(* CoDeSys 2.3 export: EXPORTEDPROJECT.EXP *)
(* Libraries: STANDARD.LIB 5.6.98 13:03:02 *)

(* Task configuration *)
TASK Standard (PRIORITY := 0, INTERVAL := T#10ms);
MAIN
END_TASK

(* POU MAIN, SFC *)
PROGRAM MAIN
VAR
	SRullo_presenza AT%IX0.0:BOOL;
	SRullo_Finecorsa AT%IX0.1:BOOL;
	SAsc_Altezza AT%IX0.2:BOOL;
	SRullo_Pistoneavanti AT%IX0.3:BOOL;
	SAsc_Capacitivo AT%IX0.4:BOOL;
	SAsc_Soglia AT%IX0.5:BOOL;
	SAsc_Pistonedietro AT%IX0.6:BOOL;
	SAsc_Basso AT%IX0.7:BOOL;
	SAsc_Alto AT%IX0.8:BOOL;
         SGiostra_Colore AT %IX0.9:BOOL;
	SGiostra_Altezza AT%IX1.0:BOOL;
	SGiostra_PresenzaPinza AT%IX1.1:BOOL;
	SDremel_alto AT%IX1.2:BOOL;
	SDremel_Basso AT %IX1.3:BOOL;
	SGiostra_Presenza AT %IX1.4:BOOL;
	SGiostra_AltezzaAlto AT %IX1.5:BOOL;
	SGiostra_AltezzaBasso AT %IX1.6:BOOL;
	SGiostra_MarkerAlto AT%IX1.7: BOOL;
	SGiostra_MarkerBasso AT%IX1.8: BOOL;



	AAsc_salita AT%QX0.0:BOOL;
	AAsc_discesa AT%QX0.1:BOOL;
	AAsc_aria AT%QX0.2:BOOL;
	AAsc_pistone AT %QX0.3:BOOL;
	ARullo_pistone AT %QX0.4:BOOL;
	ARullo_avanti AT %QX0.5:BOOL;
	AGiostra_Pistone AT %QX0.6:BOOL;
	AGiostra_Marker AT%QX4.0:BOOL;
	AGiostra_Gira AT %QX0.8:BOOL;
	AGiostra_Scarta AT%QX2.9:BOOL;
         AGiostra_Dremel AT%QX1.3:BOOL;
	AGiostra_AbbassaDremel AT%QX1.1:BOOL;
	AGiostra_Altezza AT%QX1.2:BOOL;

	S_RC_FineCorsaBasso AT %IX8.0:BOOL;
	S_RC_FineCorsaAlto AT %IX8.1:BOOL;
	S_RC_FineCorsaDestra AT %IX8.2:BOOL;
	S_RC_FineCorsaSinistra AT %IX8.3:BOOL;
	S_RC_PresenzaPinza AT %IX8.4:BOOL;
	S_RC_PinzaSensore AT %IX8.5:BOOL;
	S_RC_ScivoloPieno AT %IX8.7:BOOL;

	S_RC_Encoder AT %IX8.6:BOOL;
	S_RC_Estensimetro AT %IW2:WORD;

	A_RC_MovBasso AT %QX8.0:BOOL;
	A_RC_MovAlto AT %QX8.1:BOOL;
	A_RC_MovDestra AT %QX8.2:BOOL;
	A_RC_MovSinistra AT %QX8.3:BOOL;
	A_RC_Pinza AT %QX8.4:BOOL;

	T1: TON;
	T2: TON;
	T3: TON;
	T4: TON;
	T5: TON;
	T6: TON;
	T7: TON;
	T8: TON;
	T9: TON;
	T10: TON;
	T11: TON;
	T12: TON;
	T13: TON;
	T14: TON;
	T15: TON;
	T16: TON;
	T17: TON;
	T18: TON;
	T19: TON;

	Scarto1: BOOL;
	tra1: BOOL;
	tra2: BOOL;
	PezzoOK: BOOL;
	GiostraOK: BOOL;
	L: BOOL;
	ColoreOK: BOOL;
	P1C1B0: BOOL;
	P1C0B0: BOOL;
	L0: BOOL;
	L1: BOOL;
	L2: BOOL;
	L3: BOOL;
	L4: BOOL;
	L5: BOOL;
	L6: BOOL;
	NonRosso: BOOL;
	T: BOOL;
	Tra: BOOL;
	Rosso: BOOL;
	TrapanoOK: BOOL;
	P0C1B0: BOOL;
	P2C1B0: BOOL;
	P2C0B0: BOOL;
	Aspetta: BOOL;
	Timer: BOOL;
	P2nonRosso: BOOL;
	aspetta2: BOOL;
	P3C0B0: BOOL;
	Bucare: BOOL;
	P3C1B1: BOOL;
	TastatoreOK: BOOL;
	Vestiti: BOOL;
	NonVestiti: BOOL;
	Tast2: BOOL;
	Tast1: BOOL;
	P4C0B0: BOOL;
	MarkerOK: BOOL;
	Bucato: BOOL;
	NonBucato: BOOL;
	P4C1B1R: BOOL;
	P4C1B1W: BOOL;
	x: BOOL;
	xa: BOOL;
	xb: BOOL;
	xc: BOOL;
	Colora: BOOL;
	NonColora: BOOL;
	P5C0B0: BOOL;
	EspelliOK: BOOL;
	P5C1B1W: BOOL;
	NonColoraR: BOOL;
	P5C1B1R: BOOL;
	ScartoOK: BOOL;
	Nonscartare: BOOL;
	P6C1B1R: BOOL;
	Espelli: BOOL;
	FineGiro: BOOL;
	Robot: BOOL;
	RobotOK: BOOL;
	P7: BOOL;
	att: BOOL;
	NC: BOOL;
	Tempo: BOOL;
	TTrapano: BOOL;
	TTastatore: BOOL;
	TMarker: BOOL;
	TScarto: BOOL;
	Temsdsdpo: BOOL;
	C1: CTUD;
	Count: INT;
	RulloVuoto: BOOL;
	VarOFF: BOOL;
	VarON: BOOL;
	T20: TON;
	T21: TON;
	T22: TON;
	trans4: BOOL;
	trans6: BOOL;
	trans3: BOOL;
	T31: TON;
	T32: TON;
	T33: TON;
	T34: TON;
	T35: TON;
	T36: TON;
	T37: TON;
	T38: TON;
	T39: TON;

	UP:BOOL;
	DOWN:BOOL;
	Peso1: BOOL;
	Peso2: BOOL;
	CounterRC1: CTUD;
	POS: INT;
	V:BOOL;

	T24: TON;

	PinzaBasso: BOOL;
	IST:DINT;
	AltScivolo: BOOL;
	AltFinale: BOOL;
	SbloccoDx: BOOL;
	Z: WORD;
	Z1: STRING;
	Z2: STRING;
	Z3: DINT;
	T30: TON;
	AltBase: BOOL;
	AltBilancia: BOOL;
	Start: BOOL;
	Sali: BOOL;
	Scendi: BOOL;
	StopSali: BOOL;
	StopScendi: BOOL;
	RSD: BOOL;
	RAB: BOOL;
	BilanciaOK: BOOL;
	Scivolo3OK: BOOL;
	Scivolo2: BOOL;
	Scivolo1: BOOL;
	Scivolo3: BOOL;
	Bilancia: BOOL;
	Partenza: BOOL;
	Peso3: BOOL;
	T40: TON;
	T43: TON;
	T44: TON;
	Start1: BOOL;
	T45: TON;
	T46: TON;
	T47: TON;
	T48: TON;
	X2: STRING;
	X1: WORD;
	X3: STRING;

	SbloccoUp: BOOL;
	LBilancia: BOOL;
	L7: BOOL;
	T49: TON;
	T50: TON;
END_VAR
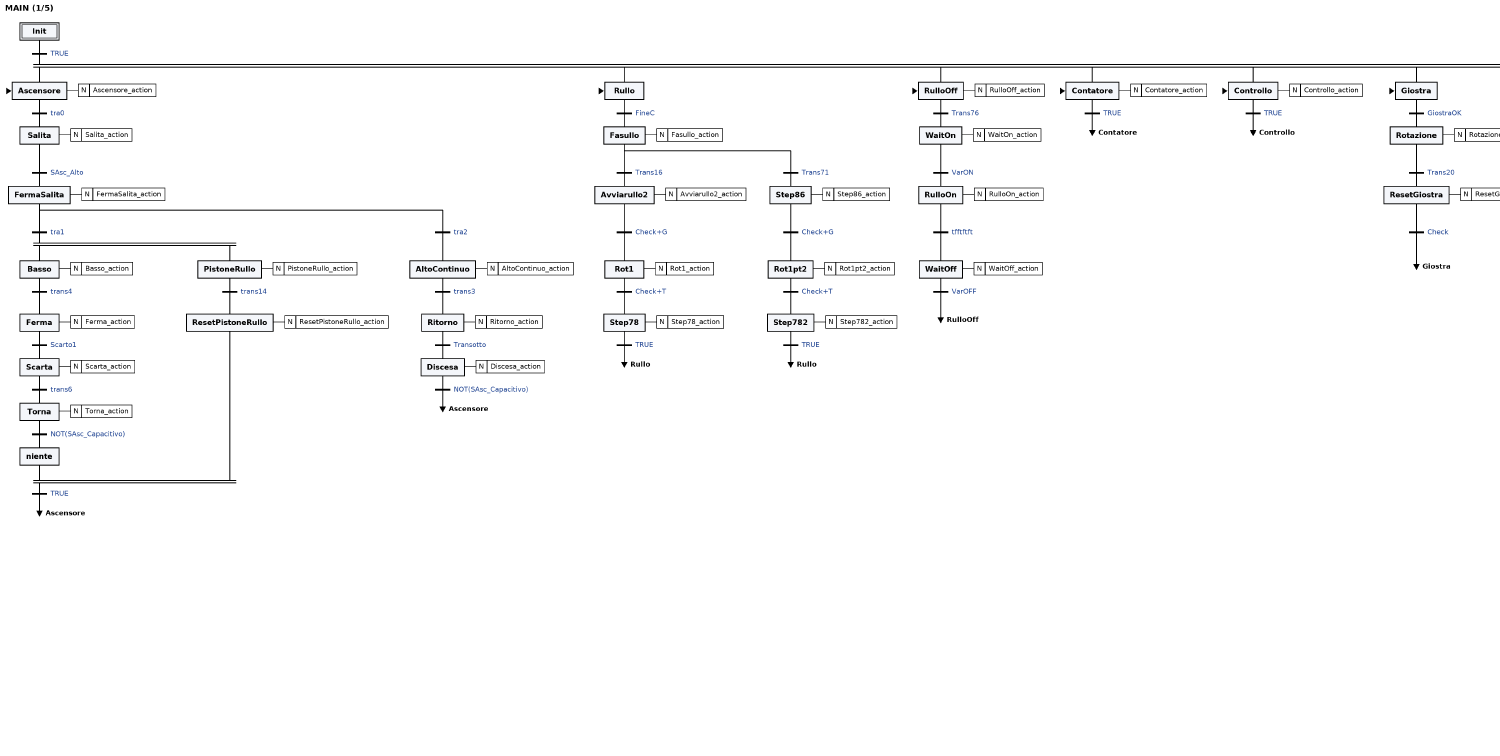
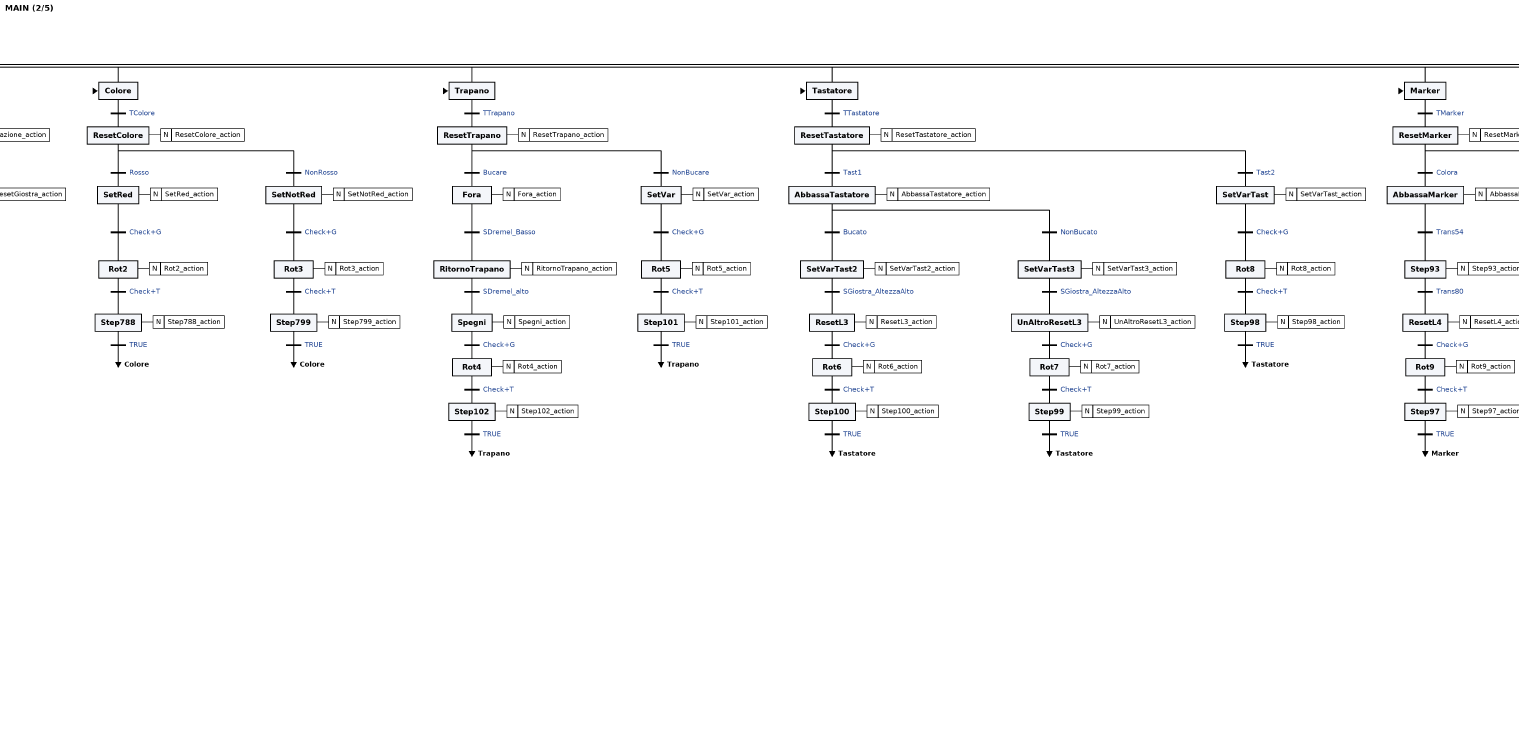
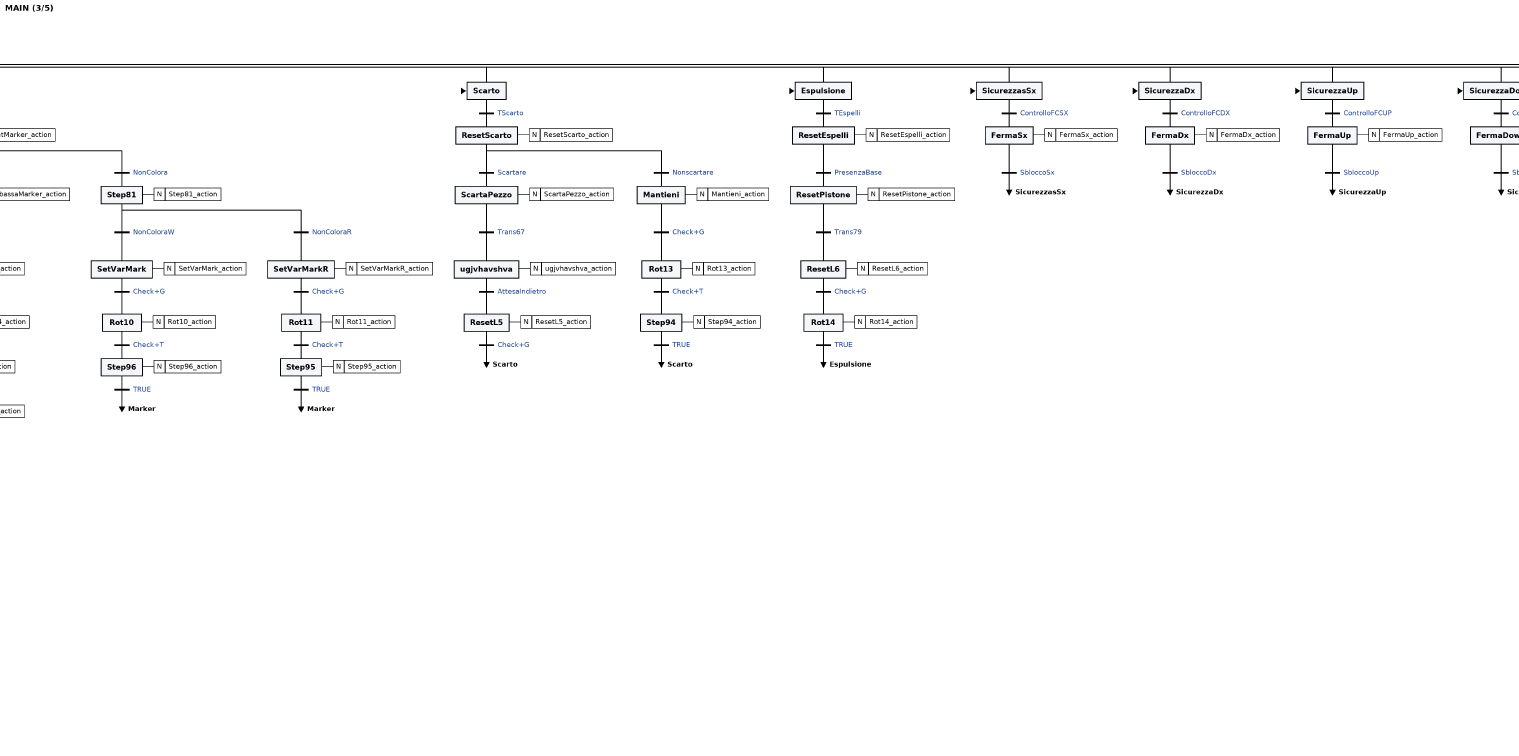
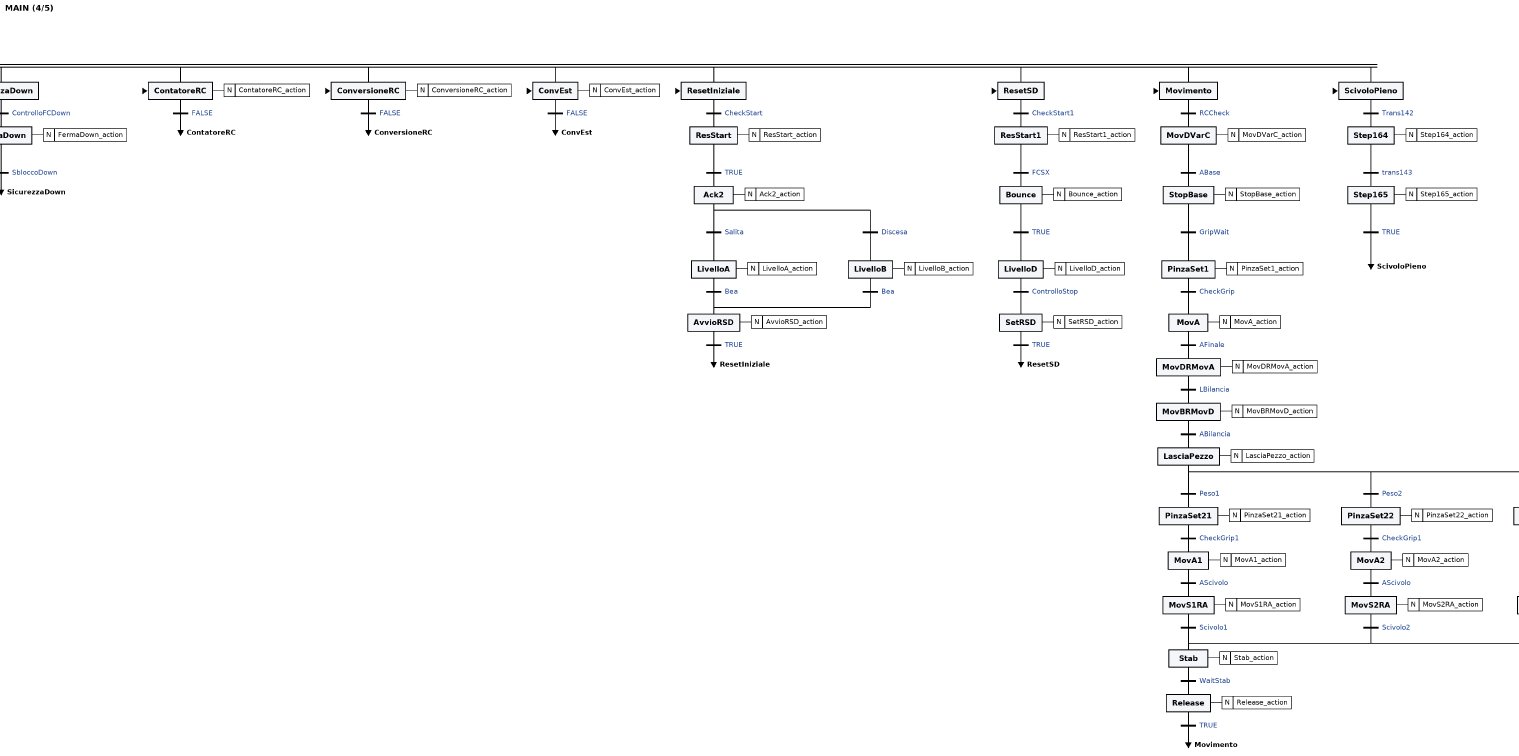
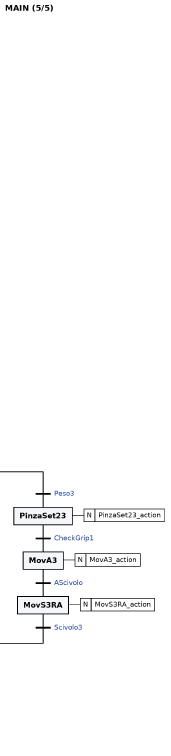
INITIAL_STEP Init:
END_STEP
TRANSITION FROM Init TO (Ascensore, Rullo, RulloOff, Contatore, Controllo, Giostra, Colore, Trapano, Tastatore, Marker, Scarto, Espulsione, SicurezzasSx, SicurezzaDx, SicurezzaUp, SicurezzaDown, ContatoreRC, ConversioneRC, ConvEst, ResetIniziale, ResetSD, Movimento, ScivoloPieno) := TRUE;
END_TRANSITION
STEP Ascensore:
	Ascensore_action(N);
END_STEP
TRANSITION FROM Ascensore TO Salita := tra0;
END_TRANSITION
STEP Salita:
	Salita_action(N);
END_STEP
TRANSITION FROM Salita TO FermaSalita := SAsc_Alto;
END_TRANSITION
STEP FermaSalita:
	FermaSalita_action(N);
END_STEP
TRANSITION FROM FermaSalita TO (Basso, PistoneRullo) := tra1;
END_TRANSITION
TRANSITION FROM FermaSalita TO AltoContinuo := tra2;
END_TRANSITION
STEP Basso:
	Basso_action(N);
END_STEP
TRANSITION FROM Basso TO Ferma := trans4;
END_TRANSITION
STEP Ferma:
	Ferma_action(N);
END_STEP
TRANSITION FROM Ferma TO Scarta := Scarto1;
END_TRANSITION
STEP Scarta:
	Scarta_action(N);
END_STEP
TRANSITION FROM Scarta TO Torna := trans6;
END_TRANSITION
STEP Torna:
	Torna_action(N);
END_STEP
TRANSITION FROM Torna TO niente := NOT(SAsc_Capacitivo);
END_TRANSITION
STEP niente:
END_STEP
STEP PistoneRullo:
	PistoneRullo_action(N);
END_STEP
TRANSITION FROM PistoneRullo TO ResetPistoneRullo := trans14;
END_TRANSITION
STEP ResetPistoneRullo:
	ResetPistoneRullo_action(N);
END_STEP
TRANSITION FROM (niente, ResetPistoneRullo) TO Ascensore := TRUE;
END_TRANSITION
STEP AltoContinuo:
	AltoContinuo_action(N);
END_STEP
TRANSITION FROM AltoContinuo TO Ritorno := trans3;
END_TRANSITION
STEP Ritorno:
	Ritorno_action(N);
END_STEP
TRANSITION FROM Ritorno TO Discesa := Transotto;
END_TRANSITION
STEP Discesa:
	Discesa_action(N);
END_STEP
TRANSITION FROM Discesa TO Ascensore := NOT(SAsc_Capacitivo);
END_TRANSITION
STEP Rullo:
END_STEP
TRANSITION FROM Rullo TO Fasullo := FineC;
END_TRANSITION
STEP RulloOff:
	RulloOff_action(N);
END_STEP
TRANSITION FROM RulloOff TO WaitOn := Trans76;
END_TRANSITION
STEP WaitOn:
	WaitOn_action(N);
END_STEP
TRANSITION FROM WaitOn TO RulloOn := VarON;
END_TRANSITION
STEP RulloOn:
	RulloOn_action(N);
END_STEP
TRANSITION FROM RulloOn TO WaitOff := tfftftft;
END_TRANSITION
STEP WaitOff:
	WaitOff_action(N);
END_STEP
TRANSITION FROM WaitOff TO RulloOff := VarOFF;
END_TRANSITION
STEP Contatore:
	Contatore_action(N);
END_STEP
TRANSITION FROM Contatore TO Contatore := TRUE;
END_TRANSITION
STEP Controllo:
	Controllo_action(N);
END_STEP
TRANSITION FROM Controllo TO Controllo := TRUE;
END_TRANSITION
STEP Fasullo:
	Fasullo_action(N);
END_STEP
TRANSITION FROM Fasullo TO Avviarullo2 := Trans16;
END_TRANSITION
TRANSITION FROM Fasullo TO Step86 := Trans71;
END_TRANSITION
STEP Avviarullo2:
	Avviarullo2_action(N);
END_STEP
TRANSITION FROM Avviarullo2 TO Rot1 := Check+G;
END_TRANSITION
STEP Step86:
	Step86_action(N);
END_STEP
TRANSITION FROM Step86 TO Rot1pt2 := Check+G;
END_TRANSITION
STEP Rot1pt2:
	Rot1pt2_action(N);
END_STEP
TRANSITION FROM Rot1pt2 TO Step782 := Check+T;
END_TRANSITION
STEP Step782:
	Step782_action(N);
END_STEP
TRANSITION FROM Step782 TO Rullo := TRUE;
END_TRANSITION
STEP Rot1:
	Rot1_action(N);
END_STEP
TRANSITION FROM Rot1 TO Step78 := Check+T;
END_TRANSITION
STEP Step78:
	Step78_action(N);
END_STEP
TRANSITION FROM Step78 TO Rullo := TRUE;
END_TRANSITION
STEP Giostra:
END_STEP
TRANSITION FROM Giostra TO Rotazione := GiostraOK;
END_TRANSITION
STEP Rotazione:
	Rotazione_action(N);
END_STEP
TRANSITION FROM Rotazione TO ResetGiostra := Trans20;
END_TRANSITION
STEP ResetGiostra:
	ResetGiostra_action(N);
END_STEP
TRANSITION FROM ResetGiostra TO Giostra := Check;
END_TRANSITION
STEP Colore:
END_STEP
TRANSITION FROM Colore TO ResetColore := TColore;
END_TRANSITION
STEP ResetColore:
	ResetColore_action(N);
END_STEP
TRANSITION FROM ResetColore TO SetRed := Rosso;
END_TRANSITION
TRANSITION FROM ResetColore TO SetNotRed := NonRosso;
END_TRANSITION
STEP SetRed:
	SetRed_action(N);
END_STEP
TRANSITION FROM SetRed TO Rot2 := Check+G;
END_TRANSITION
STEP Rot2:
	Rot2_action(N);
END_STEP
TRANSITION FROM Rot2 TO Step788 := Check+T;
END_TRANSITION
STEP Step788:
	Step788_action(N);
END_STEP
TRANSITION FROM Step788 TO Colore := TRUE;
END_TRANSITION
STEP SetNotRed:
	SetNotRed_action(N);
END_STEP
TRANSITION FROM SetNotRed TO Rot3 := Check+G;
END_TRANSITION
STEP Rot3:
	Rot3_action(N);
END_STEP
TRANSITION FROM Rot3 TO Step799 := Check+T;
END_TRANSITION
STEP Step799:
	Step799_action(N);
END_STEP
TRANSITION FROM Step799 TO Colore := TRUE;
END_TRANSITION
STEP Trapano:
END_STEP
TRANSITION FROM Trapano TO ResetTrapano := TTrapano;
END_TRANSITION
STEP ResetTrapano:
	ResetTrapano_action(N);
END_STEP
TRANSITION FROM ResetTrapano TO Fora := Bucare;
END_TRANSITION
TRANSITION FROM ResetTrapano TO SetVar := NonBucare;
END_TRANSITION
STEP Fora:
	Fora_action(N);
END_STEP
TRANSITION FROM Fora TO RitornoTrapano := SDremel_Basso;
END_TRANSITION
STEP RitornoTrapano:
	RitornoTrapano_action(N);
END_STEP
TRANSITION FROM RitornoTrapano TO Spegni := SDremel_alto;
END_TRANSITION
STEP Spegni:
	Spegni_action(N);
END_STEP
TRANSITION FROM Spegni TO Rot4 := Check+G;
END_TRANSITION
STEP Rot4:
	Rot4_action(N);
END_STEP
TRANSITION FROM Rot4 TO Step102 := Check+T;
END_TRANSITION
STEP Step102:
	Step102_action(N);
END_STEP
TRANSITION FROM Step102 TO Trapano := TRUE;
END_TRANSITION
STEP SetVar:
	SetVar_action(N);
END_STEP
TRANSITION FROM SetVar TO Rot5 := Check+G;
END_TRANSITION
STEP Rot5:
	Rot5_action(N);
END_STEP
TRANSITION FROM Rot5 TO Step101 := Check+T;
END_TRANSITION
STEP Step101:
	Step101_action(N);
END_STEP
TRANSITION FROM Step101 TO Trapano := TRUE;
END_TRANSITION
STEP Tastatore:
END_STEP
TRANSITION FROM Tastatore TO ResetTastatore := TTastatore;
END_TRANSITION
STEP ResetTastatore:
	ResetTastatore_action(N);
END_STEP
TRANSITION FROM ResetTastatore TO AbbassaTastatore := Tast1;
END_TRANSITION
TRANSITION FROM ResetTastatore TO SetVarTast := Tast2;
END_TRANSITION
STEP AbbassaTastatore:
	AbbassaTastatore_action(N);
END_STEP
TRANSITION FROM AbbassaTastatore TO SetVarTast2 := Bucato;
END_TRANSITION
TRANSITION FROM AbbassaTastatore TO SetVarTast3 := NonBucato;
END_TRANSITION
STEP SetVarTast2:
	SetVarTast2_action(N);
END_STEP
TRANSITION FROM SetVarTast2 TO ResetL3 := SGiostra_AltezzaAlto;
END_TRANSITION
STEP ResetL3:
	ResetL3_action(N);
END_STEP
TRANSITION FROM ResetL3 TO Rot6 := Check+G;
END_TRANSITION
STEP Rot6:
	Rot6_action(N);
END_STEP
TRANSITION FROM Rot6 TO Step100 := Check+T;
END_TRANSITION
STEP Step100:
	Step100_action(N);
END_STEP
TRANSITION FROM Step100 TO Tastatore := TRUE;
END_TRANSITION
STEP SetVarTast3:
	SetVarTast3_action(N);
END_STEP
TRANSITION FROM SetVarTast3 TO UnAltroResetL3 := SGiostra_AltezzaAlto;
END_TRANSITION
STEP UnAltroResetL3:
	UnAltroResetL3_action(N);
END_STEP
TRANSITION FROM UnAltroResetL3 TO Rot7 := Check+G;
END_TRANSITION
STEP Rot7:
	Rot7_action(N);
END_STEP
TRANSITION FROM Rot7 TO Step99 := Check+T;
END_TRANSITION
STEP Step99:
	Step99_action(N);
END_STEP
TRANSITION FROM Step99 TO Tastatore := TRUE;
END_TRANSITION
STEP SetVarTast:
	SetVarTast_action(N);
END_STEP
TRANSITION FROM SetVarTast TO Rot8 := Check+G;
END_TRANSITION
STEP Rot8:
	Rot8_action(N);
END_STEP
TRANSITION FROM Rot8 TO Step98 := Check+T;
END_TRANSITION
STEP Step98:
	Step98_action(N);
END_STEP
TRANSITION FROM Step98 TO Tastatore := TRUE;
END_TRANSITION
STEP Marker:
END_STEP
TRANSITION FROM Marker TO ResetMarker := TMarker;
END_TRANSITION
STEP ResetMarker:
	ResetMarker_action(N);
END_STEP
TRANSITION FROM ResetMarker TO AbbassaMarker := Colora;
END_TRANSITION
TRANSITION FROM ResetMarker TO Step81 := NonColora;
END_TRANSITION
STEP Step81:
	Step81_action(N);
END_STEP
TRANSITION FROM Step81 TO SetVarMark := NonColoraW;
END_TRANSITION
TRANSITION FROM Step81 TO SetVarMarkR := NonColoraR;
END_TRANSITION
STEP SetVarMarkR:
	SetVarMarkR_action(N);
END_STEP
TRANSITION FROM SetVarMarkR TO Rot11 := Check+G;
END_TRANSITION
STEP Rot11:
	Rot11_action(N);
END_STEP
TRANSITION FROM Rot11 TO Step95 := Check+T;
END_TRANSITION
STEP Step95:
	Step95_action(N);
END_STEP
TRANSITION FROM Step95 TO Marker := TRUE;
END_TRANSITION
STEP SetVarMark:
	SetVarMark_action(N);
END_STEP
TRANSITION FROM SetVarMark TO Rot10 := Check+G;
END_TRANSITION
STEP Rot10:
	Rot10_action(N);
END_STEP
TRANSITION FROM Rot10 TO Step96 := Check+T;
END_TRANSITION
STEP Step96:
	Step96_action(N);
END_STEP
TRANSITION FROM Step96 TO Marker := TRUE;
END_TRANSITION
STEP AbbassaMarker:
	AbbassaMarker_action(N);
END_STEP
TRANSITION FROM AbbassaMarker TO Step93 := Trans54;
END_TRANSITION
STEP Step93:
	Step93_action(N);
END_STEP
TRANSITION FROM Step93 TO ResetL4 := Trans80;
END_TRANSITION
STEP ResetL4:
	ResetL4_action(N);
END_STEP
TRANSITION FROM ResetL4 TO Rot9 := Check+G;
END_TRANSITION
STEP Rot9:
	Rot9_action(N);
END_STEP
TRANSITION FROM Rot9 TO Step97 := Check+T;
END_TRANSITION
STEP Step97:
	Step97_action(N);
END_STEP
TRANSITION FROM Step97 TO Marker := TRUE;
END_TRANSITION
STEP Scarto:
END_STEP
TRANSITION FROM Scarto TO ResetScarto := TScarto;
END_TRANSITION
STEP ResetScarto:
	ResetScarto_action(N);
END_STEP
TRANSITION FROM ResetScarto TO ScartaPezzo := Scartare;
END_TRANSITION
TRANSITION FROM ResetScarto TO Mantieni := Nonscartare;
END_TRANSITION
STEP ScartaPezzo:
	ScartaPezzo_action(N);
END_STEP
TRANSITION FROM ScartaPezzo TO ugjvhavshva := Trans67;
END_TRANSITION
STEP ugjvhavshva:
	ugjvhavshva_action(N);
END_STEP
TRANSITION FROM ugjvhavshva TO ResetL5 := AttesaIndietro;
END_TRANSITION
STEP ResetL5:
	ResetL5_action(N);
END_STEP
TRANSITION FROM ResetL5 TO Scarto := Check+G;
END_TRANSITION
STEP Mantieni:
	Mantieni_action(N);
END_STEP
TRANSITION FROM Mantieni TO Rot13 := Check+G;
END_TRANSITION
STEP Rot13:
	Rot13_action(N);
END_STEP
TRANSITION FROM Rot13 TO Step94 := Check+T;
END_TRANSITION
STEP Step94:
	Step94_action(N);
END_STEP
TRANSITION FROM Step94 TO Scarto := TRUE;
END_TRANSITION
STEP Espulsione:
END_STEP
TRANSITION FROM Espulsione TO ResetEspelli := TEspelli;
END_TRANSITION
STEP SicurezzasSx:
END_STEP
TRANSITION FROM SicurezzasSx TO FermaSx := ControlloFCSX;
END_TRANSITION
STEP FermaSx:
	FermaSx_action(N);
END_STEP
TRANSITION FROM FermaSx TO SicurezzasSx := SbloccoSx;
END_TRANSITION
STEP SicurezzaDx:
END_STEP
TRANSITION FROM SicurezzaDx TO FermaDx := ControlloFCDX;
END_TRANSITION
STEP FermaDx:
	FermaDx_action(N);
END_STEP
TRANSITION FROM FermaDx TO SicurezzaDx := SbloccoDx;
END_TRANSITION
STEP SicurezzaUp:
END_STEP
TRANSITION FROM SicurezzaUp TO FermaUp := ControlloFCUP;
END_TRANSITION
STEP SicurezzaDown:
END_STEP
TRANSITION FROM SicurezzaDown TO FermaDown := ControlloFCDown;
END_TRANSITION
STEP FermaDown:
	FermaDown_action(N);
END_STEP
TRANSITION FROM FermaDown TO SicurezzaDown := SbloccoDown;
END_TRANSITION
STEP ContatoreRC:
	ContatoreRC_action(N);
END_STEP
TRANSITION FROM ContatoreRC TO ContatoreRC := FALSE;
END_TRANSITION
STEP ConversioneRC:
	ConversioneRC_action(N);
END_STEP
TRANSITION FROM ConversioneRC TO ConversioneRC := FALSE;
END_TRANSITION
STEP ConvEst:
	ConvEst_action(N);
END_STEP
TRANSITION FROM ConvEst TO ConvEst := FALSE;
END_TRANSITION
STEP ResetIniziale:
END_STEP
TRANSITION FROM ResetIniziale TO ResStart := CheckStart;
END_TRANSITION
STEP ResStart:
	ResStart_action(N);
END_STEP
TRANSITION FROM ResStart TO Ack2 := TRUE;
END_TRANSITION
STEP Ack2:
	Ack2_action(N);
END_STEP
TRANSITION FROM Ack2 TO LivelloA := Salita;
END_TRANSITION
TRANSITION FROM Ack2 TO LivelloB := Discesa;
END_TRANSITION
STEP LivelloA:
	LivelloA_action(N);
END_STEP
TRANSITION FROM LivelloA TO AvvioRSD := Bea;
END_TRANSITION
STEP LivelloB:
	LivelloB_action(N);
END_STEP
TRANSITION FROM LivelloB TO AvvioRSD := Bea;
END_TRANSITION
STEP AvvioRSD:
	AvvioRSD_action(N);
END_STEP
TRANSITION FROM AvvioRSD TO ResetIniziale := TRUE;
END_TRANSITION
STEP ResetSD:
END_STEP
TRANSITION FROM ResetSD TO ResStart1 := CheckStart1;
END_TRANSITION
STEP ResStart1:
	ResStart1_action(N);
END_STEP
TRANSITION FROM ResStart1 TO Bounce := FCSX;
END_TRANSITION
STEP Bounce:
	Bounce_action(N);
END_STEP
TRANSITION FROM Bounce TO LivelloD := TRUE;
END_TRANSITION
STEP LivelloD:
	LivelloD_action(N);
END_STEP
TRANSITION FROM LivelloD TO SetRSD := ControlloStop;
END_TRANSITION
STEP SetRSD:
	SetRSD_action(N);
END_STEP
TRANSITION FROM SetRSD TO ResetSD := TRUE;
END_TRANSITION
STEP Movimento:
END_STEP
TRANSITION FROM Movimento TO MovDVarC := RCCheck;
END_TRANSITION
STEP ScivoloPieno:
END_STEP
TRANSITION FROM ScivoloPieno TO Step164 := Trans142;
END_TRANSITION
STEP Step164:
	Step164_action(N);
END_STEP
TRANSITION FROM Step164 TO Step165 := trans143;
END_TRANSITION
STEP Step165:
	Step165_action(N);
END_STEP
TRANSITION FROM Step165 TO ScivoloPieno := TRUE;
END_TRANSITION
STEP MovDVarC:
	MovDVarC_action(N);
END_STEP
TRANSITION FROM MovDVarC TO StopBase := ABase;
END_TRANSITION
STEP StopBase:
	StopBase_action(N);
END_STEP
TRANSITION FROM StopBase TO PinzaSet1 := GripWait;
END_TRANSITION
STEP PinzaSet1:
	PinzaSet1_action(N);
END_STEP
TRANSITION FROM PinzaSet1 TO MovA := CheckGrip;
END_TRANSITION
STEP MovA:
	MovA_action(N);
END_STEP
TRANSITION FROM MovA TO MovDRMovA := AFinale;
END_TRANSITION
STEP MovDRMovA:
	MovDRMovA_action(N);
END_STEP
TRANSITION FROM MovDRMovA TO MovBRMovD := LBilancia;
END_TRANSITION
STEP MovBRMovD:
	MovBRMovD_action(N);
END_STEP
TRANSITION FROM MovBRMovD TO LasciaPezzo := ABilancia;
END_TRANSITION
STEP LasciaPezzo:
	LasciaPezzo_action(N);
END_STEP
TRANSITION FROM LasciaPezzo TO PinzaSet21 := Peso1;
END_TRANSITION
TRANSITION FROM LasciaPezzo TO PinzaSet22 := Peso2;
END_TRANSITION
TRANSITION FROM LasciaPezzo TO PinzaSet23 := Peso3;
END_TRANSITION
STEP PinzaSet21:
	PinzaSet21_action(N);
END_STEP
TRANSITION FROM PinzaSet21 TO MovA1 := CheckGrip1;
END_TRANSITION
STEP MovA1:
	MovA1_action(N);
END_STEP
TRANSITION FROM MovA1 TO MovS1RA := AScivolo;
END_TRANSITION
STEP MovS1RA:
	MovS1RA_action(N);
END_STEP
TRANSITION FROM MovS1RA TO Stab := Scivolo1;
END_TRANSITION
STEP PinzaSet22:
	PinzaSet22_action(N);
END_STEP
TRANSITION FROM PinzaSet22 TO MovA2 := CheckGrip1;
END_TRANSITION
STEP MovA2:
	MovA2_action(N);
END_STEP
TRANSITION FROM MovA2 TO MovS2RA := AScivolo;
END_TRANSITION
STEP MovS2RA:
	MovS2RA_action(N);
END_STEP
TRANSITION FROM MovS2RA TO Stab := Scivolo2;
END_TRANSITION
STEP PinzaSet23:
	PinzaSet23_action(N);
END_STEP
TRANSITION FROM PinzaSet23 TO MovA3 := CheckGrip1;
END_TRANSITION
STEP MovA3:
	MovA3_action(N);
END_STEP
TRANSITION FROM MovA3 TO MovS3RA := AScivolo;
END_TRANSITION
STEP MovS3RA:
	MovS3RA_action(N);
END_STEP
TRANSITION FROM MovS3RA TO Stab := Scivolo3;
END_TRANSITION
STEP Stab:
	Stab_action(N);
END_STEP
TRANSITION FROM Stab TO Release := WaitStab;
END_TRANSITION
STEP Release:
	Release_action(N);
END_STEP
TRANSITION FROM Release TO Movimento := TRUE;
END_TRANSITION
STEP FermaUp:
	FermaUp_action(N);
END_STEP
TRANSITION FROM FermaUp TO SicurezzaUp := SbloccoUp;
END_TRANSITION
STEP ResetEspelli:
	ResetEspelli_action(N);
END_STEP
TRANSITION FROM ResetEspelli TO ResetPistone := PresenzaBase;
END_TRANSITION
STEP ResetPistone:
	ResetPistone_action(N);
END_STEP
TRANSITION FROM ResetPistone TO ResetL6 := Trans79;
END_TRANSITION
STEP ResetL6:
	ResetL6_action(N);
END_STEP
TRANSITION FROM ResetL6 TO Rot14 := Check+G;
END_TRANSITION
STEP Rot14:
	Rot14_action(N);
END_STEP
TRANSITION FROM Rot14 TO Espulsione := TRUE;
END_TRANSITION

ACTION Ascensore_action:
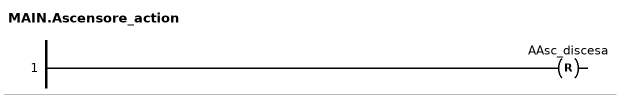
_LD_ (* Ladder Diagram *)
NETWORK 1
	* --- (R AAsc_discesa)
_END_LD_
(* the same logic as Structured Text *)
(* Network 1 *)
AAsc_discesa := FALSE;
END_ACTION

ACTION Salita_action:
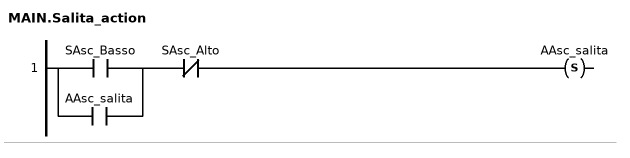
_LD_ (* Ladder Diagram *)
NETWORK 1
	{ [SAsc_Basso] | [AAsc_salita] } - [/SAsc_Alto] --- (S AAsc_salita)
_END_LD_
(* the same logic as Structured Text *)
(* Network 1 *)
IF (SAsc_Basso OR AAsc_salita) AND NOT SAsc_Alto THEN AAsc_salita := TRUE; END_IF;
END_ACTION

ACTION FermaSalita_action:
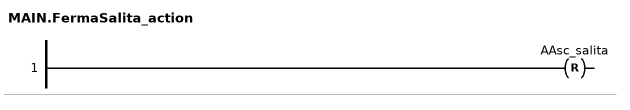
_LD_ (* Ladder Diagram *)
NETWORK 1
	* --- (R AAsc_salita)
_END_LD_
(* the same logic as Structured Text *)
(* Network 1 *)
AAsc_salita := FALSE;
END_ACTION

ACTION Basso_action:
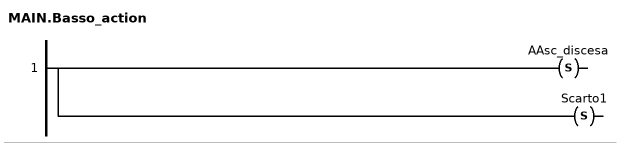
_LD_ (* Ladder Diagram *)
NETWORK 1
	* --- (S AAsc_discesa) (S Scarto1)
_END_LD_
(* the same logic as Structured Text *)
(* Network 1 *)
AAsc_discesa := TRUE;
Scarto1 := TRUE;
END_ACTION

ACTION Ferma_action:
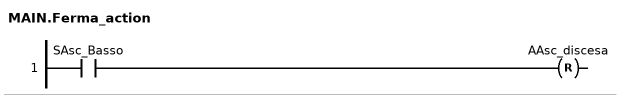
_LD_ (* Ladder Diagram *)
NETWORK 1
	[SAsc_Basso] --- (R AAsc_discesa)
_END_LD_
(* the same logic as Structured Text *)
(* Network 1 *)
IF SAsc_Basso THEN AAsc_discesa := FALSE; END_IF;
END_ACTION

ACTION Scarta_action:
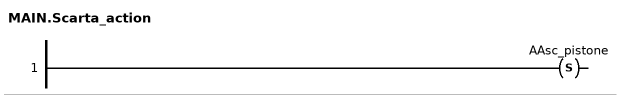
_LD_ (* Ladder Diagram *)
NETWORK 1
	* --- (S AAsc_pistone)
_END_LD_
(* the same logic as Structured Text *)
(* Network 1 *)
AAsc_pistone := TRUE;
END_ACTION

ACTION Torna_action:
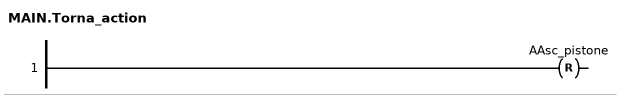
_LD_ (* Ladder Diagram *)
NETWORK 1
	* --- (R AAsc_pistone)
_END_LD_
(* the same logic as Structured Text *)
(* Network 1 *)
AAsc_pistone := FALSE;
END_ACTION

ACTION PistoneRullo_action:
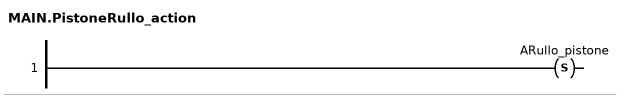
_LD_ (* Ladder Diagram *)
NETWORK 1
	* --- (S ARullo_pistone)
_END_LD_
(* the same logic as Structured Text *)
(* Network 1 *)
ARullo_pistone := TRUE;
END_ACTION

ACTION ResetPistoneRullo_action:
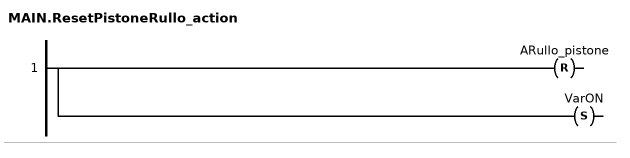
_LD_ (* Ladder Diagram *)
NETWORK 1
	* --- (R ARullo_pistone) (S VarON)
_END_LD_
(* the same logic as Structured Text *)
(* Network 1 *)
ARullo_pistone := FALSE;
VarON := TRUE;
END_ACTION

ACTION AltoContinuo_action:
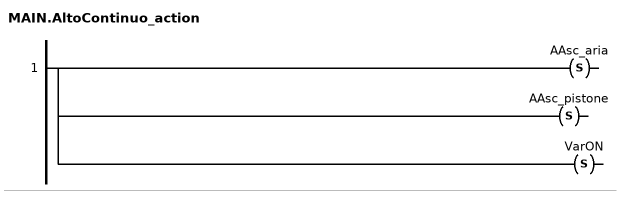
_LD_ (* Ladder Diagram *)
NETWORK 1
	* --- (S AAsc_aria) (S AAsc_pistone) (S VarON)
_END_LD_
(* the same logic as Structured Text *)
(* Network 1 *)
AAsc_aria := TRUE;
AAsc_pistone := TRUE;
VarON := TRUE;
END_ACTION

ACTION Ritorno_action:
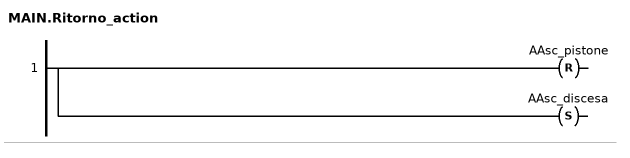
_LD_ (* Ladder Diagram *)
NETWORK 1
	* --- (R AAsc_pistone) (S AAsc_discesa)
_END_LD_
(* the same logic as Structured Text *)
(* Network 1 *)
AAsc_pistone := FALSE;
AAsc_discesa := TRUE;
END_ACTION

ACTION Discesa_action:
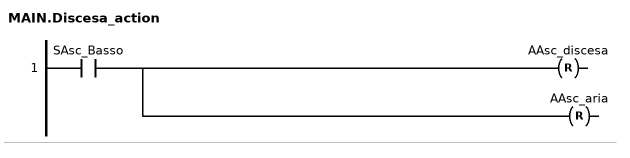
_LD_ (* Ladder Diagram *)
NETWORK 1
	[SAsc_Basso] --- (R AAsc_discesa) (R AAsc_aria)
_END_LD_
(* the same logic as Structured Text *)
(* Network 1 *)
IF SAsc_Basso THEN AAsc_discesa := FALSE; AAsc_aria := FALSE; END_IF;
END_ACTION

ACTION RulloOff_action:
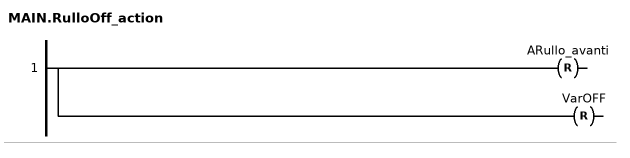
_LD_ (* Ladder Diagram *)
NETWORK 1
	* --- (R ARullo_avanti) (R VarOFF)
_END_LD_
(* the same logic as Structured Text *)
(* Network 1 *)
ARullo_avanti := FALSE;
VarOFF := FALSE;
END_ACTION

ACTION WaitOn_action:
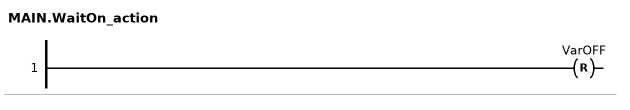
_LD_ (* Ladder Diagram *)
NETWORK 1
	* --- (R VarOFF)
_END_LD_
(* the same logic as Structured Text *)
(* Network 1 *)
VarOFF := FALSE;
END_ACTION

ACTION RulloOn_action:
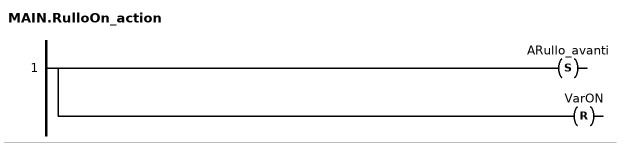
_LD_ (* Ladder Diagram *)
NETWORK 1
	* --- (S ARullo_avanti) (R VarON)
_END_LD_
(* the same logic as Structured Text *)
(* Network 1 *)
ARullo_avanti := TRUE;
VarON := FALSE;
END_ACTION

ACTION WaitOff_action:
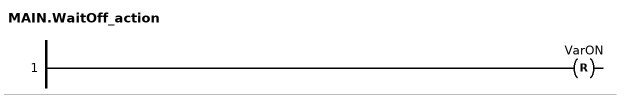
_LD_ (* Ladder Diagram *)
NETWORK 1
	* --- (R VarON)
_END_LD_
(* the same logic as Structured Text *)
(* Network 1 *)
VarON := FALSE;
END_ACTION

ACTION Contatore_action:
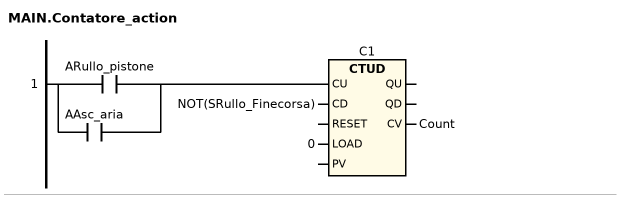
_LD_ (* Ladder Diagram *)
NETWORK 1
	{ [ARullo_pistone] | [AAsc_aria] } - C1:CTUD(CU: *, CD: NOT(SRullo_Finecorsa), RESET: , LOAD: 0, PV: , CV => Count)
_END_LD_
END_ACTION

ACTION Controllo_action:
IF Count<>0 THEN RulloVuoto:=TRUE;
ELSE RulloVuoto:=FALSE;
END_IF;
END_ACTION

ACTION Fasullo_action:
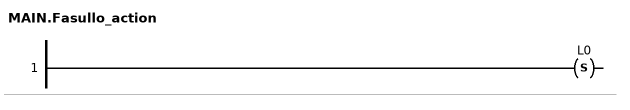
_LD_ (* Ladder Diagram *)
NETWORK 1
	* --- (S L0)
_END_LD_
(* the same logic as Structured Text *)
(* Network 1 *)
L0 := TRUE;
END_ACTION

ACTION Avviarullo2_action:
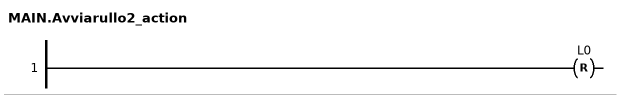
_LD_ (* Ladder Diagram *)
NETWORK 1
	* --- (R L0)
_END_LD_
(* the same logic as Structured Text *)
(* Network 1 *)
L0 := FALSE;
END_ACTION

ACTION Step86_action:
